(* IEC 61131-3 sources: DYN_pipeless_plant/PLC Data/PLC, 5 files *)

(* ---- sys_flag_types.IEC ---- *)
(*@PROPERTIES_EX@
TYPE: DATA_TYPE
LOCALE: 0
*)
TYPE
      Task_Name_Typ : ARRAY[0..9] OF BYTE;

      Extended_Task_Info   : STRUCT
      TaskName          : Task_Name_Typ;  (* Name of the Task as ARRAY OF BYTE, NULL terminated *)
      TaskPrio          : INT;            (* Priority of the task *)
      undocumented_0    : INT;
      TaskPeriod        : INT;            (* Period of the task in milliseconds *)
      TaskStack         : INT;            (* Stack size of the task *)
      unused_1          : INT;
      TaskWatchdog      : INT;            (* Watchdog time in milliseconds *)
      undocumented_2    : INT;
      undocumented_3    : INT;
      undocumented_4    : INT;
      CurDuration       : INT;            (* Current task duration in ticks including preemption *)
      MinDuration       : INT;            (* Minimum task duration in ticks including preemption *)
      MaxDuration       : INT;            (* Maximum task duration in ticks including preemption *)
      undocumented_5    : INT;
      CurDelay          : INT;            (* Current task delay in ticks including preemption *)
      MinDelay          : INT;            (* Minimum task delay in ticks including preemption *)
      MaxDelay          : INT;            (* Maximum task delay in ticks including preemption *)
   END_STRUCT;
END_TYPE

TYPE
	Task_Name_eCLR : ARRAY[0..35] OF BYTE;

	Task_Info_eCLR : STRUCT
	TaskStack            : INT;            (* Stack size of the task *)
	TaskPrio             : INT;            (* Priority of the task *)
	TaskPeriod_us        : DINT;           (* Period of the task in microseconds *)
	TaskWatchdog_us      : DINT;           (* Watchdog time in microseconds *)
	TaskPeriod           : INT;            (* Period of the task in milliseconds *)
	TaskWatchdog         : INT;            (* Watchdog time in milliseconds *)
	MinDuration_us       : DINT;           (* Minimum task duration in microseconds including preemption *)
	MaxDuration_us       : DINT;           (* Maximum task duration in microseconds including preemption *)
	CurDuration_us       : DINT;           (* Current task duration in microseconds including preemption *)
	MinDelay_us          : DINT;           (* Minimum task delay in microseconds including preemption *)
	MaxDelay_us          : DINT;           (* Maximum task delay in microseconds including preemption *)
	CurDelay_us          : DINT;           (* Current task delay in microseconds including preemption *)
	MinDuration          : INT;            (* Minimum task duration in milliseconds including preemption *)
	MaxDuration          : INT;            (* Maximum task duration in milliseconds including preemption *)
	CurDuration          : INT;            (* Current task duration in milliseconds including preemption *)
	MinDelay             : INT;            (* Minimum task delay in milliseconds including preemption *)
	MaxDelay             : INT;            (* Maximum task delay in milliseconds including preemption *)
	CurDelay             : INT;            (* Current task delay in milliseconds including preemption *)
	unused_1             : DINT;
	unused_2             : DINT;
	unused_3             : DINT;
	unused_4             : DINT;
	unused_5             : DINT;
	unused_6             : DINT;
	unused_7             : DINT;
	unused_8             : DINT;
	unused_9             : DINT;
	TNameMaxSize         : INT;
	TNameSize            : INT;
	TaskName             : Task_Name_eCLR;
	END_STRUCT;
END_TYPE

TYPE
	PND_IO_32  : ARRAY[0..31]  OF BYTE;
	PND_IO_64  : ARRAY[0..63]  OF BYTE;
	PND_IO_128 : ARRAY[0..127] OF BYTE;
	PND_IO_256 : ARRAY[0..255] OF BYTE;
	PND_IO_512 : ARRAY[0..511] OF BYTE;
	Redundancy_OPC_Struct : ARRAY[0..2] OF INT;
END_TYPE

(* ---- User_Types.IEC ---- *)
(*@PROPERTIES_EX@
TYPE: DATA_TYPE
LOCALE: 0
*)
TYPE
	ARR_TCP_DATA_B_0_999 : ARRAY[0..999] OF BYTE;
END_TYPE

(* ---- Select_Position_Mix_Vert.ST ---- *)
(*@PROPERTIES_EX@
TYPE: POU
LOCALE: 0
IEC_LANGUAGE: ST
PLC_TYPE: independent
PROC_TYPE: independent
*)
(*@KEY@:DESCRIPTION*)

(*@KEY@:END_DESCRIPTION*)
FUNCTION_BLOCK Select_Position_Mix_Vert

(*Group:Default*)

VAR_INPUT
	MPosUp :	BOOL;
	MPosDown :	BOOL;
	MPos6 :	BOOL;
	MPos5 :	BOOL;
	MPos4 :	BOOL;
	MPos3 :	BOOL;
	MPos2 :	BOOL;
	MPos1 :	BOOL;
END_VAR

VAR_EXTERNAL
	Q_0_2_0_0 :	BOOL;(*Motor3 Bit1*)
	Q_0_2_0_2 :	BOOL;(*Motor3 Bit2*)
	Q_0_2_0_1 :	BOOL;(*Motor3 Bit3*)
	Q_0_2_0_3 :	BOOL;(*Motor3 Bit4*)
END_VAR

VAR_INPUT
	MStop :	BOOL;(*Stop*)
	MPosRelRobot :	BOOL;(*Release Position (Robot)*)
	MRef :	BOOL;(*Referenzfahrt*)
END_VAR

(*@KEY@: WORKSHEET
NAME: Select_Position_Mix_Vert
IEC_LANGUAGE: ST
*)
IF MPosDown=TRUE THEN;
Q_0_2_0_0:=TRUE;
Q_0_2_0_2:=FALSE;
Q_0_2_0_1:=FALSE;
Q_0_2_0_3:=FALSE;
ELSIF MPos2=TRUE THEN;
Q_0_2_0_0:=FALSE;
Q_0_2_0_2:=TRUE;
Q_0_2_0_1:=FALSE;
Q_0_2_0_3:=FALSE;
ELSIF MPos1=TRUE THEN;
Q_0_2_0_0:=TRUE;
Q_0_2_0_2:=TRUE;
Q_0_2_0_1:=FALSE;
Q_0_2_0_3:=FALSE;
ELSIF MPosUp=TRUE THEN;
Q_0_2_0_0:=FALSE;
Q_0_2_0_2:=FALSE;
Q_0_2_0_1:=TRUE;
Q_0_2_0_3:=FALSE;  (*Danke Martin*)
(*ELSIF MPos5=TRUE THEN;
Q_0_2_0_0:=TRUE;
Q_0_2_0_2:=FALSE;
Q_0_2_0_1:=TRUE;
Q_0_2_0_3:=FALSE;
ELSIF MPos6=TRUE THEN;
Q_0_2_0_0:=TRUE;
Q_0_2_0_2:=TRUE;
Q_0_2_0_1:=TRUE;
Q_0_2_0_3:=FALSE;*)
ELSIF MRef=TRUE THEN;
Q_0_2_0_0:=FALSE;
Q_0_2_0_2:=TRUE;
Q_0_2_0_1:=FALSE;
Q_0_2_0_3:=TRUE;
ELSIF MStop=TRUE THEN;
Q_0_2_0_0:=TRUE;
Q_0_2_0_2:=FALSE;
Q_0_2_0_1:=FALSE;
Q_0_2_0_3:=TRUE;
ELSIF MPosRelRobot=TRUE THEN;
Q_0_2_0_0:=TRUE;
Q_0_2_0_2:=TRUE;
Q_0_2_0_1:=FALSE;
Q_0_2_0_3:=TRUE;
ELSE
Q_0_2_0_0:=FALSE;
Q_0_2_0_2:=FALSE;
Q_0_2_0_1:=FALSE;
Q_0_2_0_3:=FALSE;
END_IF;
(*@KEY@: END_WORKSHEET *)
END_FUNCTION_BLOCK

(* ---- Select_Position_Strg_Hor.ST ---- *)
(*@PROPERTIES_EX@
TYPE: POU
LOCALE: 0
IEC_LANGUAGE: ST
PLC_TYPE: independent
PROC_TYPE: independent
*)
(*@KEY@:DESCRIPTION*)

(*@KEY@:END_DESCRIPTION*)
FUNCTION_BLOCK Select_Position_Strg_Hor

(*Group:Default*)

VAR_INPUT
	SHPos6 :	BOOL;
	SHPos5 :	BOOL;
	SHPos2 :	BOOL;
	SHPos4 :	BOOL;
	SHPosGap :	BOOL;
	SHPos3 :	BOOL;
	SHPos1 :	BOOL;
END_VAR

VAR_EXTERNAL
	Q_0_1_0_4 :	BOOL;(*Motor1 Bit1*)
	Q_0_1_0_6 :	BOOL;(*Motor1 Bit2*)
	Q_0_1_0_5 :	BOOL;(*Motor1 Bit3*)
	Q_0_1_0_7 :	BOOL;(*Motor1 Bit4*)
END_VAR

VAR_INPUT
	SHRef :	BOOL;(*Referenzfahrt*)
	SHStop :	BOOL;(*Stop*)
END_VAR

(*@KEY@: WORKSHEET
NAME: Select_Position_Strg_Hor
IEC_LANGUAGE: ST
*)
IF SHPos1=TRUE THEN;
Q_0_1_0_4:=TRUE;
Q_0_1_0_6:=FALSE;
Q_0_1_0_5:=FALSE;
Q_0_1_0_7:=FALSE;
ELSIF SHPos2=TRUE THEN;
Q_0_1_0_4:=FALSE;
Q_0_1_0_6:=TRUE;
Q_0_1_0_5:=FALSE;
Q_0_1_0_7:=FALSE;
ELSIF SHPos3=TRUE THEN;
Q_0_1_0_4:=TRUE;
Q_0_1_0_6:=TRUE;
Q_0_1_0_5:=FALSE;
Q_0_1_0_7:=FALSE;
ELSIF SHPosGap=TRUE THEN;
Q_0_1_0_4:=FALSE;
Q_0_1_0_6:=FALSE;
Q_0_1_0_5:=TRUE;
Q_0_1_0_7:=FALSE;
ELSIF SHPos4=TRUE THEN;
Q_0_1_0_4:=TRUE;
Q_0_1_0_6:=FALSE;
Q_0_1_0_5:=TRUE;
Q_0_1_0_7:=FALSE;
ELSIF SHPos5=TRUE THEN;
Q_0_1_0_4:=FALSE;
Q_0_1_0_6:=TRUE;
Q_0_1_0_5:=TRUE;
Q_0_1_0_7:=FALSE;
ELSIF SHPos6=TRUE THEN;
Q_0_1_0_4:=TRUE;
Q_0_1_0_6:=TRUE;
Q_0_1_0_5:=TRUE;
Q_0_1_0_7:=FALSE;
ELSIF SHStop=TRUE THEN;
Q_0_1_0_4:=FALSE;
Q_0_1_0_6:=FALSE;
Q_0_1_0_5:=FALSE;
Q_0_1_0_7:=TRUE;
ELSIF SHRef=TRUE THEN;
Q_0_1_0_4:=TRUE;
Q_0_1_0_6:=FALSE;
Q_0_1_0_5:=FALSE;
Q_0_1_0_7:=TRUE;
ELSE
Q_0_1_0_4:=FALSE;
Q_0_1_0_6:=FALSE;
Q_0_1_0_5:=FALSE;
Q_0_1_0_7:=FALSE;
END_IF;
(*@KEY@: END_WORKSHEET *)
END_FUNCTION_BLOCK

(* ---- Select_Position_Strg_Ver.ST ---- *)
(*@PROPERTIES_EX@
TYPE: POU
LOCALE: 0
IEC_LANGUAGE: ST
PLC_TYPE: independent
PROC_TYPE: independent
*)
(*@KEY@:DESCRIPTION*)

(*@KEY@:END_DESCRIPTION*)
FUNCTION_BLOCK Select_Position_Strg_Ver

(*Group:Default*)

VAR_INPUT
	SVPosCent :	BOOL;
	SVPosDown :	BOOL;
	SVPosUp :	BOOL;
END_VAR

VAR_EXTERNAL
	Q_0_2_1_1 :	BOOL;(*Motor2 Bit1*)
	Q_0_2_1_3 :	BOOL;(*Motor2 Bit2*)
	Q_0_2_1_4 :	BOOL;(*Motor2 Bit3*)
	Q_0_2_1_6 :	BOOL;(*Motor2 Bit4*)
END_VAR

VAR_INPUT
	SVRef :	BOOL;(*ReferenzFahrt starten*)
	SVRelPl :	BOOL;(*Release Position Plate*)
	SVRelRo :	BOOL;(*Release Position Robot*)
	SVStop :	BOOL;(*Stop*)
END_VAR

(*@KEY@: WORKSHEET
NAME: Select_Position_Strg_Ver
IEC_LANGUAGE: ST
*)
IF SVPosDown=TRUE THEN;
Q_0_2_1_1:=TRUE;
Q_0_2_1_3:=FALSE;
Q_0_2_1_4:=FALSE;
Q_0_2_1_6:=FALSE;
ELSIF SVPosCent=TRUE THEN;
Q_0_2_1_1:=FALSE;
Q_0_2_1_3:=TRUE;
Q_0_2_1_4:=FALSE;
Q_0_2_1_6:=FALSE;
ELSIF SVPosUp=TRUE THEN;
Q_0_2_1_1:=TRUE;
Q_0_2_1_3:=TRUE;
Q_0_2_1_4:=FALSE;
Q_0_2_1_6:=FALSE;
ELSIF SVStop=TRUE THEN;
Q_0_2_1_1:=FALSE;
Q_0_2_1_3:=FALSE;
Q_0_2_1_4:=TRUE;
Q_0_2_1_6:=FALSE;
ELSIF SVRef=TRUE THEN;
Q_0_2_1_1:=TRUE;
Q_0_2_1_3:=FALSE;
Q_0_2_1_4:=TRUE;
Q_0_2_1_6:=FALSE;
ElSIF SVRelPl=TRUE THEN;
Q_0_2_1_1:=TRUE;
Q_0_2_1_3:=TRUE;
Q_0_2_1_4:=TRUE;
Q_0_2_1_6:=FALSE;
ElSIF SVRelRo=TRUE THEN;
Q_0_2_1_1:=FALSE;
Q_0_2_1_3:=FALSE;
Q_0_2_1_4:=FALSE;
Q_0_2_1_6:=TRUE;
ELSE (* Huefner: Adding ELSE Condition, setting all to FALSE if no position is given *)
Q_0_2_1_1:=FALSE;
Q_0_2_1_3:=FALSE;
Q_0_2_1_4:=FALSE;
Q_0_2_1_6:=FALSE;
END_IF;

(*@KEY@: END_WORKSHEET *)
END_FUNCTION_BLOCK
